VISUALIZATION visu_a20  // 2x2
END_VISUALIZATION

(* stored: Version 1.1.0.1, ProductVersion 3.1.4024.12
   Visu visu_a20: Id {0b6daab3-3e13-4e30-9bed-7d31837494f1} *)
